// TIA Portal V18 export
// export: Created 2026-01-09T11:31:56.5068031Z, ExportSetting WithDefaults, DisplayName Totally Integrated Automation Portal, DisplayVersion V18 Update 5, DisplayName TIA Portal Openness, DisplayVersion V18 Update 5, DisplayName TIA Portal Teamcenter Gateway, DisplayVersion V18, DisplayName TIA Portal Version Control Interface, DisplayVersion V18, DisplayName SINAMICS Startdrive Advanced, DisplayVersion V18 SP2 Update 1, DisplayName SINAMICS Startdrive G110M, G120, G120C, G120D, G120P, G115D, DisplayVersion V18 SP2 Update 1, DisplayName SINAMICS Startdrive G130, G150, S120, S150, SINAMICS MV, S210, G220, S200, DisplayVersion V18 SP2 Update 1, DisplayName STEP 7 Professional, DisplayVersion V18 Update 5, DisplayName STEP 7 Safety, DisplayVersion V18, DisplayName WinCC Professional, DisplayVersion V18 Update 5
TagTable "Glue"
  GluingControl_Input_GluingDeviceReady : Bool  (PLC tag GluingControl.Input.GluingDeviceReady, CPU S71500-2PN_TP700, 1 s)
  GluingControl_Input_GluingFault : Bool  (PLC tag GluingControl.Input.GluingFault, CPU S71500-2PN_TP700, 1 s)
  GluingControl_Input_GluingRefillTank : Bool  (PLC tag GluingControl.Input.GluingRefillTank, CPU S71500-2PN_TP700, 1 s)
  GluingControl_Input_GluingTankEmpty : Bool  (PLC tag GluingControl.Input.GluingTankEmpty, CPU S71500-2PN_TP700, 1 s)
  GluingControl_Output_GluingPro_X : Bool  (PLC tag GluingControl.Output.GluingPro_X, CPU S71500-2PN_TP700, 1 s)
  GluingControl_Output_GluingPro_Y : Bool  (PLC tag GluingControl.Output.GluingPro_Y, CPU S71500-2PN_TP700, 1 s)
  GluingControl_Output_GluingPro_Z : Bool  (PLC tag GluingControl.Output.GluingPro_Z, CPU S71500-2PN_TP700, 1 s)
  GluingControl_Output_GluingReset : Bool  (PLC tag GluingControl.Output.GluingReset, CPU S71500-2PN_TP700, 1 s)
  GluingControl_Control_Manual_X : Bool  (PLC tag GluingControl.Control.Manual_X, CPU S71500-2PN_TP700, 1 s)
  GluingControl_Control_Manual_Y : Bool  (PLC tag GluingControl.Control.Manual_Y, CPU S71500-2PN_TP700, 1 s)
  GluingControl_Control_Manual_Z : Bool  (PLC tag GluingControl.Control.Manual_Z, CPU S71500-2PN_TP700, 1 s)
  GluingControl_Control_ManualTest_X : Bool  (PLC tag GluingControl.Control.ManualTest_X, CPU S71500-2PN_TP700, 1 s)
  GluingControl_Control_ManualTestStartGlue : Bool  (PLC tag GluingControl.Control.ManualTestStartGlue, CPU S71500-2PN_TP700, 1 s)
  GluingControl_GlueCalibraton : Bool  (PLC tag GluingControl.GlueCalibratonMode, CPU S71500-2PN_TP700, 1 s)
